(*
SPDX-FileCopyrightText: © 2026 Oleksandr Tiutyk <trofimich@gmail.com>
SPDX-License-Identifier: MIT
License: https://opensource.org/license/mit
*)

(*!
<summary>
Wraps native exception codes; the manager provides a separate borrowed static view for each cyclic PLC task.
</summary>
<description>
Registered dynamic instances/clones belong to DynamicMemoryManager and must not be deleted manually. Instances
and borrowed views must not cross task boundaries. The static view changes on the next native catch in its
owning task. Framework propagation preserves the captured code, catch point and timestamps in a dynamic clone.
Implements ISystemException so handlers can query the captured native code through an interface. Root lookup
returns this instance as a borrowed read-only view. The native throw source is unknown. Messages include the
captured catch point regardless of showSource; the catch point is not the throw source. Dynamic copies are
explicitly registered by Clone after construction; plain __NEW does not transfer ownership to the task
manager.
</description>
*)

{attribute 'enable_dynamic_creation'}
{attribute 'no_explicit_call' := 'do not call this function block directly'}
FUNCTION_BLOCK SystemException EXTENDS Object IMPLEMENTS ISystemException
VAR_STAT
	//! <summary>Class name shared by all instances of this function block.</summary>
	{attribute 'hide'} 
	_ClassName : STRING := __POUNAME();
END_VAR
VAR
	{attribute 'hide'} 
	_ExceptionCode : __SYSTEM.ExceptionCode;
	_LocalTimestamp : LDATE_AND_TIME;
	_UtcTimestamp : LDATE_AND_TIME;
	{attribute 'hide'} 	
	_CatchPointNamespaceName : STRING;
	{attribute 'hide'} 
	_CatchPointPOUName : STRING;
	{attribute 'hide'} 
	_CatchPointPosition : STRING;
	
	{attribute 'hide'} 
	_UnspecifiedPOU : STRING(128);

	{attribute 'hide'} 
	_UnspecifiedPosition : STRING(32);

	
END_VAR

(*!
<summary>Appends the selected timestamp to an existing diagnostic target.</summary>
<description>
Borrows the writable diagnostic buffer for the call. Hidden mode leaves it unchanged; otherwise appends the
supplied local or UTC timestamp, with a UTC suffix for UTC mode. Passes the concrete ERROR_MESSAGE buffer
to string helpers so their descriptors retain the WSTRING type and full target capacity. Formats without
dynamic memory allocation.
</description>
*)
METHOD PRIVATE appendTimestampDescription
VAR_IN_OUT
	targetMessage : ERROR_MESSAGE;
END_VAR
VAR_INPUT
	timestampDisplayMode : TIMESTAMP_DISPLAY_MODE := TIMESTAMP_DISPLAY_MODE.HIDDEN;
	localTimestamp : LDATE_AND_TIME;	
	utcTimestamp : LDATE_AND_TIME;	
END_VAR
VAR
	targetMessagePointer : POINTER TO ERROR_MESSAGE;
END_VAR
IF timestampDisplayMode = TIMESTAMP_DISPLAY_MODE.HIDDEN THEN
	RETURN;
END_IF

targetMessagePointer := ADR(targetMessage);

CASE timestampDisplayMode OF
	TIMESTAMP_DISPLAY_MODE.LOCAL:
		WideStrings.AppendFit255(targetMessagePointer^, TO_WSTRING(localTimestamp));
	
	TIMESTAMP_DISPLAY_MODE.UTC:
		WideStrings.AppendFit255(targetMessagePointer^, TO_WSTRING(utcTimestamp), "UTC");
END_CASE
END_METHOD

{attribute 'monitoring' := 'call'}
PROPERTY ClassName : REFERENCE TO STRING
GET
ClassName REF= _ClassName;
END_GET
END_PROPERTY

(*!
<summary>Clears the code: Empty becomes TRUE and GetMessage returns an empty string.</summary>
<description>
Resets captured timestamps to LongDateAndTimes.EPOCH; does not delete/unregister the instance. Catch-point
storage is retained.
</description>
*)

METHOD Clear
_ExceptionCode := __SYSTEM.ExceptionCode.RTSEXCPT_NOEXCEPTION;
_LocalTimestamp := LongDateAndTimes.EPOCH;
_UtcTimestamp := LongDateAndTimes.EPOCH;
END_METHOD

(*!
<summary>Returns an auto-disposed copy of the code and catch point, borrowed until cleanup.</summary>
<description>
Captured timestamps are copied unchanged; cloning does not create a new occurrence time. Allocation failure
latches and raises fatal OUT_OF_MEMORY, without a heap exception. Registers the newly constructed instance
before copying payload, outside FB_init. Registration failure releases the unregistered instance and raises a
terminal error; copy failure leaves the registered instance owned by the task manager for cleanup. Custom
overrides must follow the same ownership sequence.
</description>
*)

METHOD Clone : IObject
VAR
	exceptionClone : POINTER TO SystemException;
END_VAR
DynamicMemoryManager.RaiseIfAllocationFailed();
exceptionClone := __NEW(SystemException);

IF exceptionClone = 0 THEN
	DynamicMemoryManager.RaiseAllocationFailure();
END_IF

DynamicMemoryManager.RegisterAutoDisposedObject(autoDisposedObject := exceptionClone^);

exceptionClone^._ExceptionCode := _ExceptionCode;
exceptionClone^._CatchPointNamespaceName := _CatchPointNamespaceName;
exceptionClone^._CatchPointPOUName := _CatchPointPOUName;
exceptionClone^._CatchPointPosition := _CatchPointPosition;
exceptionClone^._LocalTimestamp := _LocalTimestamp;
exceptionClone^._UtcTimestamp := _UtcTimestamp;

Clone := exceptionClone^;
END_METHOD

(*!
<summary>Captures a native exception code, catch point and observation time.</summary>
<description>
Replaces the previous code and catch-point strings with copies of the supplied values. Captures the current
task local and UTC time when GetLastException observes the exception; the original native throw time and
source are unavailable. Input references are not retained. Descendants cannot replace native exception
capture; this operation preserves the configured code, catch location and timestamps.
</description>
*)

METHOD INTERNAL FINAL Configure
VAR_IN_OUT CONSTANT
	exceptionCode : __SYSTEM.ExceptionCode;
	catchPointNamespaceName : STRING;
	catchPointPOUName : STRING;
	catchPointPosition : STRING;
END_VAR
_ExceptionCode := exceptionCode;
_CatchPointNamespaceName := catchPointNamespaceName;
_CatchPointPOUName := catchPointPOUName;
_CatchPointPosition := catchPointPosition;
_LocalTimestamp := System.SystemLocalDateTime;
_UtcTimestamp := System.SystemUtcDateTime;
END_METHOD

(*!
<summary>Reports whether no native exception code is stored.</summary>
<description>TRUE exactly when ExceptionCode is NOEXCEPTION; does not change the captured description.</description>
*)
{attribute 'monitoring' := 'call'}
PROPERTY Empty : BOOL
GET
Empty := _ExceptionCode = __SYSTEM.ExceptionCode.RTSEXCPT_NOEXCEPTION;
END_GET
END_PROPERTY

(*!
<summary>Returns the captured native exception code.</summary>
<description>Reading preserves the stored code; NOEXCEPTION represents an empty system exception.</description>
*)
{attribute 'monitoring' := 'call'}
PROPERTY FINAL ExceptionCode : __SYSTEM.ExceptionCode
GET
ExceptionCode := _ExceptionCode;
END_GET
END_PROPERTY

(*!
<summary>Initializes placeholders for unavailable native source metadata.</summary>
<description>Does not capture an exception, allocate a diagnostic exception or raise an exception.</description>
*)
METHOD FB_init : BOOL
VAR_INPUT
	bInitRetains : BOOL; // TRUE: the retain variables are initialized (reset warm / reset cold)
	bInCopyCode : BOOL;  // TRUE: the instance will be copied to the copy code afterward (online change)
END_VAR
_UnspecifiedPOU := Exceptions.UNSPECIFIED_SOURCE;
_UnspecifiedPosition := Exceptions.UNSPECIFIED_SOURCE;
END_METHOD

(*!
<summary>Describes the captured native code and the location where it was caught.</summary>
<description>
Returns an empty message for RTSEXCPT_NOEXCEPTION. Otherwise always includes the catch point, which does not
identify the unknown native throw source. Formatting does not change the captured timestamps. A result
exceeding ERROR_MESSAGE capacity retains its prefix and ends with an ellipsis instead of raising a
size-overflow exception. Formats directly into the result without heap allocation or builders.
</description>
<param name="showSource">
Has no effect: the native throw source is unavailable. The catch point remains part of the message.
</param>
<param name="timestampDisplayMode">Selects whether the captured local or UTC timestamp is appended, or hidden.</param>
*)

METHOD FINAL GetMessage : ERROR_MESSAGE
VAR_INPUT
	showSource : BOOL := FALSE;
	timestampDisplayMode : TIMESTAMP_DISPLAY_MODE := TIMESTAMP_DISPLAY_MODE.HIDDEN;
END_VAR
IF _ExceptionCode <> __SYSTEM.ExceptionCode.RTSEXCPT_NOEXCEPTION THEN
	WideStrings.AppendFit255(
		GetMessage,
		"System exception ",
		TO_WSTRING(_ExceptionCode),
		" occured. Caught in ",
		TO_WSTRING(_CatchPointNamespaceName),
		".",
		TO_WSTRING(_CatchPointPOUName),
		" at ",
		TO_WSTRING(_CatchPointPosition));
			
	IF timestampDisplayMode <> TIMESTAMP_DISPLAY_MODE.HIDDEN THEN
		WideStrings.AppendFit255(GetMessage, Exceptions.TIME_PREFIX);
		appendTimestampDescription(
	targetMessage := GetMessage,
	timestampDisplayMode := timestampDisplayMode,
	localTimestamp := LocalTimestamp,
	utcTimestamp := UtcTimestamp
);
	END_IF
ELSE
	GetMessage := "";
END_IF
END_METHOD

(*!
<summary>Returns a borrowed read-only view of the root exception.</summary>
<description>
No clone is created and ownership is not transferred. The view does not extend the exception's lifetime and
does not expose Clear.
</description>
*)

METHOD FINAL GetRootException : IReadOnlyException
GetRootException := THIS^;
END_METHOD

(*!
<summary>Formats the available exception source description.</summary>
<description>
Returns an independent bounded string. Native exceptions without original throw-site information return the
unspecified-source marker; catch-point information is not an original throw site.
</description>
*)
METHOD FINAL GetSourceDescription : STRING(255)
GetSourceDescription := Exceptions.UNSPECIFIED_SOURCE;
END_METHOD

(*!
<summary>Provides the stored local timestamp of this exception.</summary>
<description>
Framework exceptions capture it when thrown; native exceptions capture it when GetLastException obtains their
description. Cloning preserves the timestamp; reading it does not read the current clock.
</description>
*)
{attribute 'monitoring' := 'call'}
PROPERTY FINAL LocalTimestamp : LDATE_AND_TIME
GET
LocalTimestamp := _LocalTimestamp;
END_GET
END_PROPERTY

(*!
<summary>Provides the library namespace used in diagnostics.</summary>
<description>
Borrowed read-only reference to the compiler-initialized library namespace; no ownership transfer.
</description>
*)
{attribute 'monitoring' := 'call'}
PROPERTY NamespaceName : REFERENCE TO STRING
GET
NamespaceName REF= CurrentNamespace.Name;
END_GET
END_PROPERTY

(*!
<summary>Reports the byte size of this concrete instance.</summary>
<description>
Uses XSIZEOF on the instance. Does not include separately allocated payloads or prove that an arbitrary
address is valid.
</description>
*)
{attribute 'monitoring' := 'call'}
PROPERTY SelfSize : ULINT
GET
SelfSize := XSIZEOF(THIS^);
END_GET
END_PROPERTY

(*!
<summary>Reports CRITICAL severity for a native system exception.</summary>
<description>This implementation uses a fixed severity, independent of the captured native exception code.</description>
*)
{attribute 'monitoring' := 'call'}
PROPERTY FINAL Severity : ERROR_SEVERITY
GET
Severity := ERROR_SEVERITY.CRITICAL;
END_GET
END_PROPERTY

(*!
<summary>Returns a borrowed unspecified-source marker.</summary>
<description>
Native exceptions do not provide their original POU name. The reference is read-only by contract and remains
valid only while this instance exists.
</description>
*)
{attribute 'monitoring' := 'call'}
PROPERTY FINAL SourceFullPOUName : REFERENCE TO STRING(128)
GET
SourceFullPOUName REF= _UnspecifiedPOU;
END_GET
END_PROPERTY

(*!
<summary>Returns a borrowed unspecified-position marker.</summary>
<description>
Native exceptions do not provide their original throw position. The reference is read-only by contract and
remains valid only while this instance exists.
</description>
*)
{attribute 'monitoring' := 'call'}
PROPERTY FINAL SourcePosition : REFERENCE TO STRING(32)
GET
SourcePosition REF= _UnspecifiedPosition;
END_GET
END_PROPERTY

(*!
<summary>Copies exception diagnostics and timestamps into an ERROR value.</summary>
<description>
An invalid target reference is ignored. Otherwise fills both top and root descriptions from this exception
using the supplied severity and stored timestamps. Formats the source and message once each and copies the
same results into both descriptions. Formatting uses default source and timestamp display options. The target
retains copied text, not an exception reference; formatting may follow the allocation-failure policy of the
concrete formatter.
</description>
*)
METHOD ToError
VAR_IN_OUT CONSTANT
	targetError : ERROR;
END_VAR
VAR_INPUT
	severity : ERROR_SEVERITY;	
END_VAR
VAR
	topSourceText : STRING(255);
	topMessageText : ERROR_MESSAGE;
END_VAR
IF NOT __ISVALIDREF(targetError) THEN
	RETURN;
END_IF

topSourceText := GetSourceDescription();
topMessageText := GetMessage();

targetError.Fill(
	severity := severity,
	topSource := topSourceText,
	rootSource := topSourceText,
	topMessage := topMessageText,
	rootMessage := topMessageText,
	localTimestamp := LocalTimestamp,
	utcTimestamp := UtcTimestamp
);
END_METHOD

(*!
<summary>Provides the stored UTC timestamp of this exception.</summary>
<description>
Framework exceptions capture it when thrown; native exceptions capture it when GetLastException obtains their
description. Cloning preserves the timestamp; reading it does not read the current clock.
</description>
*)
{attribute 'monitoring' := 'call'}
PROPERTY FINAL UtcTimestamp : LDATE_AND_TIME
GET
UtcTimestamp := _UtcTimestamp;
END_GET
END_PROPERTY

END_FUNCTION_BLOCK

(* stored: Version 1.1.0.1
   POU SystemException: Id {003dda89-959c-4208-b47c-eab6a22da353}, SpecialFunc None
   Folder Service methods: Id {e40f07a0-bb69-43d2-9344-558beb521327}
   Method appendTimestampDescription: Id {dcf3179b-315e-43cb-bffb-a9cc08face8f}
   Property ClassName: Id {f6998750-94de-4b27-9017-ad7539ef8bae}
   Get Get: Id {cb7835e8-806f-4442-837f-895002f84c14}
   Method Clear: Id {dbd66dfc-fc8f-4256-a0f4-f74c9a16f7ea}
   Method Clone: Id {654edb60-f1ae-4e3d-854a-ef1384720f30}
   Method Configure: Id {297ea316-2fb7-4596-b05c-db0f46e37b1b}
   Property Empty: Id {038c5f5f-d26f-4e70-a390-6d5e8f198afd}
   Get Get: Id {60ffea73-58f0-48cd-a1b6-f69c50756f23}
   Property ExceptionCode: Id {98df4acc-7b54-406f-b517-a9c22c0f0d8e}
   Get Get: Id {90619a75-6b17-438b-a2b1-b465d62fd70b}
   Method FB_init: Id {9df7f179-6b56-448d-8f6f-07eac327896a}
   Method GetMessage: Id {a88a8b1a-9f6a-4c9d-9ec5-e6c280a6e922}
   Method GetRootException: Id {cfc4f0f7-35c9-4eb3-b854-bd2edbdcadfe}
   Method GetSourceDescription: Id {933b59e0-81e6-42d6-ba36-d2e00c47553a}
   Property LocalTimestamp: Id {243bf917-8856-414f-8657-d2ad403ee832}
   Get Get: Id {79d470da-f79a-4a33-bf4f-89aa38c370f7}
   Property NamespaceName: Id {ca510274-b070-4a45-bc4b-9eb8a5a40ec1}
   Get Get: Id {6c4acd0f-2e61-4a39-b5a8-d3f83794230d}
   Property SelfSize: Id {45a123fb-1e78-493d-ab14-ef856a5a55f6}
   Get Get: Id {adba8c9d-7fbf-47a5-ad28-a9aff99bf348}
   Property Severity: Id {5e42d487-fb84-4ef7-8167-9ccf2b832212}
   Get Get: Id {deb70a32-6e78-47a9-8646-53719a2a7ac5}
   Property SourceFullPOUName: Id {bb5b4681-7cbe-4420-8da3-3eab8d25b3a6}
   Get Get: Id {000c96a6-91dd-487f-a89a-7a0a528ae1fc}
   Property SourcePosition: Id {a0036bdf-f7b1-4700-90c9-8ba4e7777c8e}
   Get Get: Id {81eb6bc3-98ea-458a-b91b-7e4c86ab7dcc}
   Method ToError: Id {5bcd52e5-ca90-49d6-b86c-fe61de2dd705}
   Property UtcTimestamp: Id {b9a20ffe-1a2b-4d8b-a985-efb4f4570353}
   Get Get: Id {9ac21bad-7080-4914-9567-5b68982f14d9} *)
